KUKA KRL program: ab_com_02_st01_g01.src, ab_com_02_st01_g01.dat

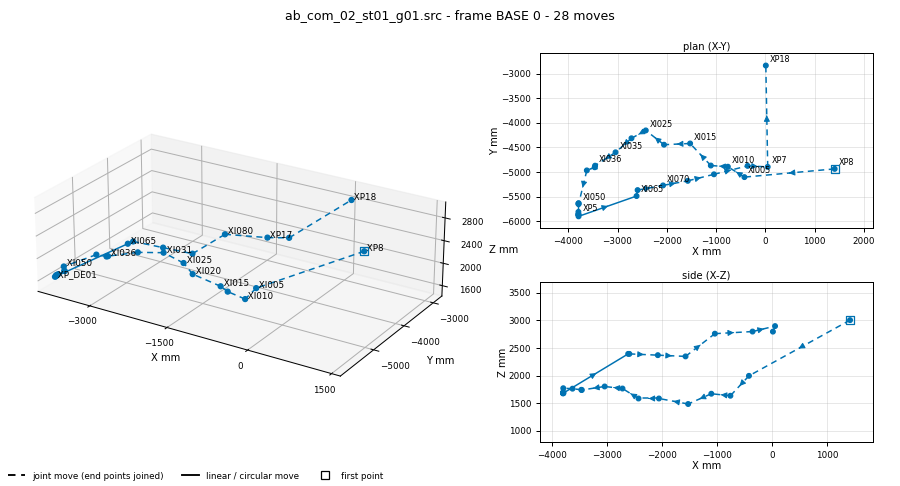
[picture p0: tool path of ab_com_02_st01_g01.src in frame BASE 0, 28 of 28 moves have a stored position in this frame; points joined in program order, loops and branches not executed]
--- ab_com_02_st01_g01.src ---
&ACCESS RVO4
&REL 783
&COMMENT Deposita axor atego 903 geo
&PARAM DISKPATH = KRC:\R1\Program\MANIPULACAO NTC
&PARAM TEMPLATE = C:\KRC\Roboter\Template\vorgabe
&PARAM EDITMASK = *
DEF AB_COM_02_ST01_G01 ( )
;FOLD INI
  ;FOLD BASISTECH INI
    GLOBAL INTERRUPT DECL 3 WHEN $STOPMESS==TRUE DO IR_STOPM ( )
    INTERRUPT ON 3
    BAS (#INITMOV,0)
  ;ENDFOLD (BASISTECH INI)
;FOLD GRIPPERTECH INI
USER_GRP(0,DUMMY,DUMMY,GDEFAULT)
;ENDFOLD (GRIPPERTECH INI)
  ;FOLD USER INI
    ;Make your modifications here

  ;ENDFOLD (USER INI)
;ENDFOLD (INI)

; Caracterizacao dos meios de producao
; Changes: Deposita Traseira LTA/LTB
; Versao Atual: 05/01/2016
; Ferramenta: Gripper 903
; Name: P13.050-R1

chk_w9_wechs_ok ( ) ;CHECK GRIPPER 903

;FOLD PTP P8 Vel=50 % PDAT7 Tool[10]:Grp 903 c/ pc Base[0];%{PE}%R 8.2.20,%MKUKATPBASIS,%CMOVE,%VPTP,%P 1:PTP, 2:P8, 3:, 5:50, 7:PDAT7
$BWDSTART=FALSE
PDAT_ACT=PPDAT7
FDAT_ACT=FP8
BAS(#PTP_PARAMS,50)
PTP XP8
;ENDFOLD

; LIGA INTERTRAVAMENTO 2 C/ R2 GARRA
;FOLD Collision.Monitoring_2_On ;%{PE}%MKUKATPUSER
COLLSTOP( 2, 1 ) ;Interrupt-Controlled
;ENDFOLD

; LIGA INTERTRAVAMENTO 3 C/ R3 GARRA
;FOLD Collision.Monitoring_3_On ;%{PE}%MKUKATPUSER
COLLSTOP( 3, 1 ) ;Interrupt-Controlled
;ENDFOLD

; LIGA INTERTRAVAMENTO 4 C/ R4 GARRA
;FOLD Collision.Monitoring_4_On ;%{PE}%MKUKATPUSER
COLLSTOP( 4, 1 ) ;Interrupt-Controlled
;ENDFOLD

; LIGA INTERTRAVAMENTO 5 C/ R5 GARRA
;FOLD Collision.Monitoring_5_On ;%{PE}%MKUKATPUSER
COLLSTOP( 5, 1 ) ;not Interrupt-Controlled
;ENDFOLD


;FOLD PTP l005 CONT Vel=50 % P_OLP2 Tool[10]:Grp 903 c/ pc Base[0];%{PE}%R 8.2.20,%MKUKATPBASIS,%CMOVE,%VPTP,%P 1:PTP, 2:l005, 3:C_DIS, 5:50, 7:P_OLP2
$BWDSTART=FALSE
PDAT_ACT=PP_OLP2
FDAT_ACT=Fl005
BAS(#PTP_PARAMS,50)
PTP Xl005 C_DIS
;ENDFOLD
;FOLD PTP l010 CONT Vel=50 % P_OLP3 Tool[10]:Grp 903 c/ pc Base[0];%{PE}%R 8.2.20,%MKUKATPBASIS,%CMOVE,%VPTP,%P 1:PTP, 2:l010, 3:C_DIS, 5:50, 7:P_OLP3
$BWDSTART=FALSE
PDAT_ACT=PP_OLP3
FDAT_ACT=Fl010
BAS(#PTP_PARAMS,50)
PTP Xl010 C_DIS
;ENDFOLD

;AGUARDA LIBERACAO DE ENTRADA
;FOLD OUT 3348 'Fora area GEOBOX' State=TRUE ;%{PE}%R 8.2.20,%MKUKATPBASIS,%COUT,%VOUTX,%P 2:3348, 3:Fora area GEOBOX, 5:TRUE, 6:
$OUT[3348]=TRUE
;ENDFOLD
;FOLD OUT 3369 'RB -PLC Interlock' State=TRUE ;%{PE}%R 8.2.20,%MKUKATPBASIS,%COUT,%VOUTX,%P 2:3369, 3:RB -PLC Interlock, 5:TRUE, 6:
$OUT[3369]=TRUE
;ENDFOLD
;FOLD WAIT FOR ( IN 3369 'RB-PLC interlocks' );%{PE}%R 8.2.20,%MKUKATPBASIS,%CEXT_WAIT_FOR,%VEXT_WAIT_FOR,%P 2:, 4:, 5:$IN, 6:3369, 7:RB-PLC interlocks, 9:
WAIT FOR  ( $IN[3369] )
;ENDFOLD
;FOLD OUT 3369 'RB -PLC Interlock' State=FALSE ;%{PE}%R 8.2.20,%MKUKATPBASIS,%COUT,%VOUTX,%P 2:3369, 3:RB -PLC Interlock, 5:FALSE, 6:
$OUT[3369]=FALSE
;ENDFOLD
;FOLD OUT 3348 'Fora area GEOBOX' State=FALSE ;%{PE}%R 8.2.20,%MKUKATPBASIS,%COUT,%VOUTX,%P 2:3348, 3:Fora area GEOBOX, 5:FALSE, 6:
$OUT[3348]=FALSE
;ENDFOLD

;FOLD PTP pp1 CONT Vel=50 % PDAT4 Tool[10]:Grp 903 c/ pc Base[0];%{PE}%R 8.2.20,%MKUKATPBASIS,%CMOVE,%VPTP,%P 1:PTP, 2:pp1, 3:C_DIS, 5:50, 7:PDAT4
$BWDSTART=FALSE
PDAT_ACT=PPDAT4
FDAT_ACT=Fpp1
BAS(#PTP_PARAMS,50)
PTP Xpp1 C_DIS
;ENDFOLD
;FOLD PTP l015 CONT Vel=50 % P_OLP4 Tool[10]:Grp 903 c/ pc Base[0];%{PE}%R 8.2.20,%MKUKATPBASIS,%CMOVE,%VPTP,%P 1:PTP, 2:l015, 3:C_DIS, 5:50, 7:P_OLP4
$BWDSTART=FALSE
PDAT_ACT=PP_OLP4
FDAT_ACT=Fl015
BAS(#PTP_PARAMS,50)
PTP Xl015 C_DIS
;ENDFOLD
;FOLD PTP l020 CONT Vel=50 % P_OLP5 Tool[10]:Grp 903 c/ pc Base[0];%{PE}%R 8.2.20,%MKUKATPBASIS,%CMOVE,%VPTP,%P 1:PTP, 2:l020, 3:C_DIS, 5:50, 7:P_OLP5
$BWDSTART=FALSE
PDAT_ACT=PP_OLP5
FDAT_ACT=Fl020
BAS(#PTP_PARAMS,50)
PTP Xl020 C_DIS
;ENDFOLD
;FOLD PTP l025 CONT Vel=50 % P_OLP6 Tool[10]:Grp 903 c/ pc Base[0];%{PE}%R 8.2.20,%MKUKATPBASIS,%CMOVE,%VPTP,%P 1:PTP, 2:l025, 3:C_DIS, 5:50, 7:P_OLP6
$BWDSTART=FALSE
PDAT_ACT=PP_OLP6
FDAT_ACT=Fl025
BAS(#PTP_PARAMS,50)
PTP Xl025 C_DIS
;ENDFOLD
;FOLD PTP l031 CONT Vel=50 % P_OLP15 Tool[10]:Grp 903 c/ pc Base[0];%{PE}%R 8.2.20,%MKUKATPBASIS,%CMOVE,%VPTP,%P 1:PTP, 2:l031, 3:C_DIS, 5:50, 7:P_OLP15
$BWDSTART=FALSE
PDAT_ACT=PP_OLP15
FDAT_ACT=Fl031
BAS(#PTP_PARAMS,50)
PTP Xl031 C_DIS
;ENDFOLD
;FOLD PTP l035 CONT Vel=50 % P_OLP8 Tool[10]:Grp 903 c/ pc Base[0];%{PE}%R 8.2.20,%MKUKATPBASIS,%CMOVE,%VPTP,%P 1:PTP, 2:l035, 3:C_DIS, 5:50, 7:P_OLP8
$BWDSTART=FALSE
PDAT_ACT=PP_OLP8
FDAT_ACT=Fl035
BAS(#PTP_PARAMS,50)
PTP Xl035 C_DIS
;ENDFOLD
;FOLD PTP l036 CONT Vel=50 % P_OLP16 Tool[10]:Grp 903 c/ pc Base[0];%{PE}%R 8.2.20,%MKUKATPBASIS,%CMOVE,%VPTP,%P 1:PTP, 2:l036, 3:C_DIS, 5:50, 7:P_OLP16
$BWDSTART=FALSE
PDAT_ACT=PP_OLP16
FDAT_ACT=Fl036
BAS(#PTP_PARAMS,50)
PTP Xl036 C_DIS
;ENDFOLD

;AGUARDA LIBERACAO PARA DEPOSITO
;FOLD OUT 3374 'Lib. Dep. Axor/Atego' State=TRUE ;%{PE}%R 8.2.20,%MKUKATPBASIS,%COUT,%VOUTX,%P 2:3374, 3:Lib. Dep. Axor/Atego, 5:TRUE, 6:
$OUT[3374]=TRUE
;ENDFOLD
;FOLD OUT 3372 'Lib. pré Dep. Axor/Atego' State=TRUE ;%{PE}%R 8.2.20,%MKUKATPBASIS,%COUT,%VOUTX,%P 2:3372, 3:Lib. pré Dep. Axor/Atego, 5:TRUE, 6:
$OUT[3372]=TRUE
;ENDFOLD
;FOLD WAIT FOR ( IN 3372 'Lib. pré Deposito Axor/Atego' );%{PE}%R 8.2.20,%MKUKATPBASIS,%CEXT_WAIT_FOR,%VEXT_WAIT_FOR,%P 2:, 4:, 5:$IN, 6:3372, 7:Lib. pré Deposito Axor/Atego, 9:
WAIT FOR  ( $IN[3372] )
;ENDFOLD
;FOLD OUT 3372 'Lib. pré Dep. Axor/Atego' State=FALSE ;%{PE}%R 8.2.20,%MKUKATPBASIS,%COUT,%VOUTX,%P 2:3372, 3:Lib. pré Dep. Axor/Atego, 5:FALSE, 6:
$OUT[3372]=FALSE
;ENDFOLD
;FOLD OUT 3374 'Lib. Dep. Axor/Atego' State=FALSE ;%{PE}%R 8.2.20,%MKUKATPBASIS,%COUT,%VOUTX,%P 2:3374, 3:Lib. Dep. Axor/Atego, 5:FALSE, 6:
$OUT[3374]=FALSE
;ENDFOLD

;FOLD PTP l040 CONT Vel=50 % P_OLP9 Tool[10]:Grp 903 c/ pc Base[0];%{PE}%R 8.2.20,%MKUKATPBASIS,%CMOVE,%VPTP,%P 1:PTP, 2:l040, 3:C_DIS, 5:50, 7:P_OLP9
$BWDSTART=FALSE
PDAT_ACT=PP_OLP9
FDAT_ACT=Fl040
BAS(#PTP_PARAMS,50)
PTP Xl040 C_DIS
;ENDFOLD
;FOLD PTP l045 CONT Vel=50 % PDAT1 Tool[10]:Grp 903 c/ pc Base[0];%{PE}%R 8.2.20,%MKUKATPBASIS,%CMOVE,%VPTP,%P 1:PTP, 2:l045, 3:C_DIS, 5:50, 7:PDAT1
$BWDSTART=FALSE
PDAT_ACT=PPDAT1
FDAT_ACT=Fl045
BAS(#PTP_PARAMS,50)
PTP Xl045 C_DIS
;ENDFOLD

; POSICAO DE VERIFICACAO DE VENTOSA OK
;FOLD PTP l050 Vel=50 % P_OLP10 Tool[10]:Grp 903 c/ pc Base[0];%{PE}%R 8.2.20,%MKUKATPBASIS,%CMOVE,%VPTP,%P 1:PTP, 2:l050, 3:, 5:50, 7:P_OLP10
$BWDSTART=FALSE
PDAT_ACT=PP_OLP10
FDAT_ACT=Fl050
BAS(#PTP_PARAMS,50)
PTP Xl050
;ENDFOLD

IF (NOT(GHOST())) THEN
chk_w9_grp5_vac_on( )      ; VENTOSA OK
ENDIF

;FOLD PTP pp2 CONT Vel=100 % PDAT5 Tool[10]:Grp 903 c/ pc Base[0];%{PE}%R 8.2.20,%MKUKATPBASIS,%CMOVE,%VPTP,%P 1:PTP, 2:pp2, 3:C_DIS, 5:100, 7:PDAT5
$BWDSTART=FALSE
PDAT_ACT=PPDAT5
FDAT_ACT=Fpp2
BAS(#PTP_PARAMS,100)
PTP Xpp2 C_DIS
;ENDFOLD
;FOLD PTP l055 CONT Vel=100 % P_OLP11 Tool[10]:Grp 903 c/ pc Base[0];%{PE}%R 8.2.20,%MKUKATPBASIS,%CMOVE,%VPTP,%P 1:PTP, 2:l055, 3:C_DIS, 5:100, 7:P_OLP11
$BWDSTART=FALSE
PDAT_ACT=PP_OLP11
FDAT_ACT=Fl055
BAS(#PTP_PARAMS,100)
PTP Xl055 C_DIS
;ENDFOLD
;FOLD LIN P9 CONT Vel=0.5 m/s CPDAT8 Tool[10]:Grp 903 c/ pc Base[0];%{PE}%R 8.2.20,%MKUKATPBASIS,%CMOVE,%VLIN,%P 1:LIN, 2:P9, 3:C_DIS C_DIS, 5:0.5, 7:CPDAT8
$BWDSTART=FALSE
LDAT_ACT=LCPDAT8
FDAT_ACT=FP9
BAS(#CP_PARAMS,0.5)
LIN XP9 C_DIS C_DIS
;ENDFOLD

; ABRE GRAMPOS INFERIORES P/ ENCAIXAR NA GEOBOX
; TECLA DE ESTADO "7"
;FOLD SET Z1.1/2 GRP AXOR 903 State=OPN GDAT1;%{PE}%R 8.2.1,%MKUKATPGRP,%CGRP,%VGRP,%P 2:7, 4:1, 5:#NO, 6:GDAT1, 8:0, 10:0
H50(GRP,7,1,GGDAT1)
;ENDFOLD
chk_w9_grp1_opn( )

;FOLD LIN P5 CONT Vel=0.5 m/s CPDAT4 Tool[10]:Grp 903 c/ pc Base[0];%{PE}%R 8.2.20,%MKUKATPBASIS,%CMOVE,%VLIN,%P 1:LIN, 2:P5, 3:C_DIS C_DIS, 5:0.5, 7:CPDAT4
$BWDSTART=FALSE
LDAT_ACT=LCPDAT4
FDAT_ACT=FP5
BAS(#CP_PARAMS,0.5)
LIN XP5 C_DIS C_DIS
;ENDFOLD
;FOLD LIN P14 CONT Vel=0.5 m/s CPDAT13 Tool[10]:Grp 903 c/ pc Base[0];%{PE}%R 8.2.20,%MKUKATPBASIS,%CMOVE,%VLIN,%P 1:LIN, 2:P14, 3:C_DIS C_DIS, 5:0.5, 7:CPDAT13
$BWDSTART=FALSE
LDAT_ACT=LCPDAT13
FDAT_ACT=FP14
BAS(#CP_PARAMS,0.5)
LIN XP14 C_DIS C_DIS
;ENDFOLD

; POSICAO DE APOIO ROLETE
;FOLD LIN P12 Vel=0.3 m/s CPDAT11 Tool[10]:Grp 903 c/ pc Base[0];%{PE}%R 8.2.20,%MKUKATPBASIS,%CMOVE,%VLIN,%P 1:LIN, 2:P12, 3:, 5:0.3, 7:CPDAT11
$BWDSTART=FALSE
LDAT_ACT=LCPDAT11
FDAT_ACT=FP12
BAS(#CP_PARAMS,0.3)
LIN XP12
;ENDFOLD

; DESLIGA INTERTRAVAMENTO 3 C/ R3 GARRA
;FOLD Collision.Monitoring_3_Off . ;%{PE}%MKUKATPUSER
COLLSTOP( 3, 2+0 )
;ENDFOLD

; DESLIGA INTERTRAVAMENTO 5 C/ R5 GARRA
;FOLD Collision.Monitoring_5_Off . ;%{PE}%MKUKATPUSER
COLLSTOP( 5, 2+0 )
;ENDFOLD

;FOLD ; Aguarda posicionamento dos Grippers R2 e R3 com rolamentos;%{PE}%R 8.2.20,%MKUKATPBASIS,%CCOMMENT,%VNORMAL,%P 2:Aguarda posicionamento dos Grippers R2 e R3 com rolamentos
;ENDFOLD
;FOLD OUT 3373 'Em pos de pre Dep AXOR/ATEGO' State=TRUE ;%{PE}%R 8.2.20,%MKUKATPBASIS,%COUT,%VOUTX,%P 2:3373, 3:Em pos de pre Dep AXOR/ATEGO, 5:TRUE, 6:
$OUT[3373]=TRUE
;ENDFOLD
;FOLD WAIT FOR ( IN 3374 'Lib. Deposito Axor/Atego' );%{PE}%R 8.2.20,%MKUKATPBASIS,%CEXT_WAIT_FOR,%VEXT_WAIT_FOR,%P 2:, 4:, 5:$IN, 6:3374, 7:Lib. Deposito Axor/Atego, 9:
WAIT FOR  ( $IN[3374] )
;ENDFOLD
;FOLD OUT 3373 'Em pos de pre Dep AXOR/ATEGO' State=FALSE ;%{PE}%R 8.2.20,%MKUKATPBASIS,%COUT,%VOUTX,%P 2:3373, 3:Em pos de pre Dep AXOR/ATEGO, 5:FALSE, 6:
$OUT[3373]=FALSE
;ENDFOLD

;FOLD ; Desliga Ventosa / Recua Cilindros / Verifica;%{PE}%R 8.2.20,%MKUKATPBASIS,%CCOMMENT,%VNORMAL,%P 2:Desliga Ventosa / Recua Cilindros / Verifica
;ENDFOLD
;FOLD SET Z6.1 VAC AXOR 903 State=BLOW GDAT26;%{PE}%R 8.2.1,%MKUKATPGRP,%CGRP,%VGRP,%P 2:13, 4:2, 5:#NO, 6:GDAT26, 8:0, 10:0
H50(GRP,13,2,GGDAT26)
;ENDFOLD
;FOLD SET Z6.1 VAC AXOR 903 State=OFF GDAT6;%{PE}%R 8.2.1,%MKUKATPGRP,%CGRP,%VGRP,%P 2:13, 4:3, 5:#NO, 6:GDAT6, 8:0, 10:0
H50(GRP,13,3,GGDAT6)
;ENDFOLD
;FOLD SET Z7.1 GRP 7 AXOR 903 State=OPN GDAT28;%{PE}%R 8.2.1,%MKUKATPGRP,%CGRP,%VGRP,%P 2:14, 4:1, 5:#NO, 6:GDAT28, 8:0, 10:0
H50(GRP,14,1,GGDAT28)
;ENDFOLD
chk_w9_grp4_opn( )
chk_w9_grp5_vac_off( )

; POSICAO DE DEPOSITO LTA/LTB
;FOLD LIN P_DE01  Vel=0.25 m/s L_OLP3 Tool[10]:Grp 903 c/ pc Base[0];%{PE}%R8.2.19,%MKUKATPBASIS,%CMOVE,%VLIN,%P 1:LIN, 2:P_DE01, 3: , 5:0.25, 7:L_OLP3
$BWDSTART = FALSE
LDAT_ACT= LL_OLP3
FDAT_ACT= FP_DE01
BAS(#CP_PARAMS,0.25)
LIN XP_DE01
;ENDFOLD

; DESLIGA INTERTRAVAMENTO 4 C/ R4 GARRA
;FOLD Collision.Monitoring_4_Off . ;%{PE}%MKUKATPUSER
COLLSTOP( 4, 2+0 )
;ENDFOLD

;FOLD OUT 3375 'Lib. p/ sair s/ Gripper Axor/Atego' State=TRUE ;%{PE}%R 8.2.20,%MKUKATPBASIS,%COUT,%VOUTX,%P 2:3375, 3:Lib. p/ sair s/ Gripper Axor/Atego, 5:TRUE, 6:
$OUT[3375]=TRUE
;ENDFOLD

; FECHA GRAMPOS INFERIORES
; TECLA DE ESTADO "7"
;FOLD SET Z1.1/2 GRP AXOR 903 State=CLO GDAT5;%{PE}%R 8.2.1,%MKUKATPGRP,%CGRP,%VGRP,%P 2:7, 4:2, 5:#NO, 6:GDAT5, 8:0, 10:0
H50(GRP,7,2,GGDAT5)
;ENDFOLD
chk_w9_grp1_clo( )

;AGUARDA LIBERACAO SAIR SEM GARRA
;FOLD OUT 3375 'Lib. p/ sair s/ Gripper Axor/Atego' State=TRUE ;%{PE}%R 8.2.20,%MKUKATPBASIS,%COUT,%VOUTX,%P 2:3375, 3:Lib. p/ sair s/ Gripper Axor/Atego, 5:TRUE, 6:
$OUT[3375]=TRUE
;ENDFOLD
;FOLD WAIT FOR ( IN 3375 'Lib. p/ sair s/ Gripper Axor/Atego' );%{PE}%R 8.2.20,%MKUKATPBASIS,%CEXT_WAIT_FOR,%VEXT_WAIT_FOR,%P 2:, 4:, 5:$IN, 6:3375, 7:Lib. p/ sair s/ Gripper Axor/Atego, 9:
WAIT FOR  ( $IN[3375] )
;ENDFOLD
;FOLD OUT 3375 'Lib. p/ sair s/ Gripper Axor/Atego' State=FALSE ;%{PE}%R 8.2.20,%MKUKATPBASIS,%COUT,%VOUTX,%P 2:3375, 3:Lib. p/ sair s/ Gripper Axor/Atego, 5:FALSE, 6:
$OUT[3375]=FALSE
;ENDFOLD

; COMANDOS PARA DESACOPLAR GRIPPER
;FOLD OUT 224 'Bloquear MPS' State=FALSE ;%{PE}%R 8.2.20,%MKUKATPBASIS,%COUT,%VOUTX,%P 2:224, 3:Bloquear MPS, 5:FALSE, 6:
$OUT[224]=FALSE
;ENDFOLD
;FOLD OUT 223 'Desbloquear MPS' State=TRUE ;%{PE}%R 8.2.20,%MKUKATPBASIS,%COUT,%VOUTX,%P 2:223, 3:Desbloquear MPS, 5:TRUE, 6:
$OUT[223]=TRUE
;ENDFOLD
;FOLD WAIT FOR ( IN 217 'MPS Destravado' );%{PE}%R 8.2.20,%MKUKATPBASIS,%CEXT_WAIT_FOR,%VEXT_WAIT_FOR,%P 2:, 4:, 5:$IN, 6:217, 7:MPS Destravado, 9:
WAIT FOR  ( $IN[217] )
;ENDFOLD
;FOLD WAIT FOR NOT ( IN 221 'MPS Travado' );%{PE}%R 8.2.20,%MKUKATPBASIS,%CEXT_WAIT_FOR,%VEXT_WAIT_FOR,%P 2:NOT, 4:, 5:$IN, 6:221, 7:MPS Travado, 9:
WAIT FOR  NOT ( $IN[221] )
;ENDFOLD
;FOLD WAIT Time=0.5 sec;%{PE}%R 8.2.20,%MKUKATPBASIS,%CWAIT,%VWAIT,%P 3:0.5
WAIT SEC 0.5
;ENDFOLD
;FOLD IBUS OFF;%{PE}%R 8.2.20,%MKUKATPBASIS,%CIBUS,%VMAP,%P 2:#OFF, 3:1
$IBUS_OFF=$IBUS_ON
$IBUS_ON=0
;ENDFOLD
;FOLD WAIT Time=0.25 sec;%{PE}%R 8.2.20,%MKUKATPBASIS,%CWAIT,%VWAIT,%P 3:0.25
WAIT SEC 0.25
;ENDFOLD

;FOLD LIN l065 Vel=0.25 m/s L_OLP4 Tool[8]:TOOL_CHANGER Base[0];%{PE}%R 8.2.20,%MKUKATPBASIS,%CMOVE,%VLIN,%P 1:LIN, 2:l065, 3:, 5:0.25, 7:L_OLP4
$BWDSTART=FALSE
LDAT_ACT=LL_OLP4
FDAT_ACT=Fl065
BAS(#CP_PARAMS,0.25)
LIN Xl065
;ENDFOLD

;FOLD WAIT FOR NOT ( IN 219 'Posicao p/ Acoplamento OK' );%{PE}%R 8.2.20,%MKUKATPBASIS,%CEXT_WAIT_FOR,%VEXT_WAIT_FOR,%P 2:NOT, 4:, 5:$IN, 6:219, 7:Posicao p/ Acoplamento OK, 9:
WAIT FOR  NOT ( $IN[219] )
;ENDFOLD
;FOLD OUT 223 'Desbloquear MPS' State=FALSE ;%{PE}%R 8.2.20,%MKUKATPBASIS,%COUT,%VOUTX,%P 2:223, 3:Desbloquear MPS, 5:FALSE, 6:
$OUT[223]=FALSE
;ENDFOLD

;FOLD LIN P2 CONT Vel=1 m/s CPDAT1 Tool[10]:Grp 903 c/ pc Base[0];%{PE}%R 8.2.20,%MKUKATPBASIS,%CMOVE,%VLIN,%P 1:LIN, 2:P2, 3:C_DIS C_DIS, 5:1, 7:CPDAT1
$BWDSTART=FALSE
LDAT_ACT=LCPDAT1
FDAT_ACT=FP2
BAS(#CP_PARAMS,1)
LIN XP2 C_DIS C_DIS
;ENDFOLD
;FOLD PTP l070 CONT Vel=100 % P_OLP12 Tool[10]:Grp 903 c/ pc Base[0];%{PE}%R 8.2.20,%MKUKATPBASIS,%CMOVE,%VPTP,%P 1:PTP, 2:l070, 3:C_DIS, 5:100, 7:P_OLP12
$BWDSTART=FALSE
PDAT_ACT=PP_OLP12
FDAT_ACT=Fl070
BAS(#PTP_PARAMS,100)
PTP Xl070 C_DIS
;ENDFOLD
;FOLD PTP l075 CONT Vel=100 % P_OLP13 Tool[10]:Grp 903 c/ pc Base[0];%{PE}%R 8.2.20,%MKUKATPBASIS,%CMOVE,%VPTP,%P 1:PTP, 2:l075, 3:C_DIS, 5:100, 7:P_OLP13
$BWDSTART=FALSE
PDAT_ACT=PP_OLP13
FDAT_ACT=Fl075
BAS(#PTP_PARAMS,100)
PTP Xl075 C_DIS
;ENDFOLD
;FOLD PTP l080 CONT Vel=100 % P_OLP14 Tool[10]:Grp 903 c/ pc Base[0];%{PE}%R 8.2.20,%MKUKATPBASIS,%CMOVE,%VPTP,%P 1:PTP, 2:l080, 3:C_DIS, 5:100, 7:P_OLP14
$BWDSTART=FALSE
PDAT_ACT=PP_OLP14
FDAT_ACT=Fl080
BAS(#PTP_PARAMS,100)
PTP Xl080 C_DIS
;ENDFOLD
;FOLD PTP P17 CONT Vel=100 % PDAT10 Tool[10]:Grp 903 c/ pc Base[0];%{PE}%R 8.2.20,%MKUKATPBASIS,%CMOVE,%VPTP,%P 1:PTP, 2:P17, 3:C_DIS, 5:100, 7:PDAT10
$BWDSTART=FALSE
PDAT_ACT=PPDAT10
FDAT_ACT=FP17
BAS(#PTP_PARAMS,100)
PTP XP17 C_DIS
;ENDFOLD

; DESLIGA INTERTRAVAMENTO 2 C/ R2 GARRA
;FOLD Collision.Monitoring_2_Off . ;%{PE}%MKUKATPUSER
COLLSTOP( 2, 2+0 )
;ENDFOLD

;LIBERA AREA
;FOLD OUT 3348 'Fora area GEOBOX' State=TRUE ;%{PE}%R 8.2.20,%MKUKATPBASIS,%COUT,%VOUTX,%P 2:3348, 3:Fora area GEOBOX, 5:TRUE, 6:
$OUT[3348]=TRUE
;ENDFOLD
;FOLD PULSE 3344 'R1 Entregou Peça GeoBox' State=TRUE Time=3 sec;%{PE}%R 8.2.20,%MKUKATPBASIS,%COUT,%VPULSE,%P 2:3344, 3:R1 Entregou Peça GeoBox, 5:TRUE, 6:, 8:3
PULSE($OUT[3344], TRUE,3)
;ENDFOLD

;FOLD PTP P7 CONT Vel=100 % PDAT6 Tool[10]:Grp 903 c/ pc Base[0];%{PE}%R 8.2.20,%MKUKATPBASIS,%CMOVE,%VPTP,%P 1:PTP, 2:P7, 3:C_DIS, 5:100, 7:PDAT6
$BWDSTART=FALSE
PDAT_ACT=PPDAT6
FDAT_ACT=FP7
BAS(#PTP_PARAMS,100)
PTP XP7 C_DIS
;ENDFOLD
;FOLD PTP P18 CONT Vel=100 % PDAT11 Tool[10]:Grp 903 c/ pc Base[0];%{PE}%R 8.2.20,%MKUKATPBASIS,%CMOVE,%VPTP,%P 1:PTP, 2:P18, 3:C_DIS, 5:100, 7:PDAT11
$BWDSTART=FALSE
PDAT_ACT=PPDAT11
FDAT_ACT=FP18
BAS(#PTP_PARAMS,100)
PTP XP18 C_DIS
;ENDFOLD

END

--- ab_com_02_st01_g01.dat ---
&ACCESS RVO4
&REL 783
&COMMENT Deposita axor atego 903 geo
&PARAM DISKPATH = KRC:\R1\Program\MANIPULACAO NTC
&PARAM TEMPLATE = C:\KRC\Roboter\Template\vorgabe
&PARAM EDITMASK = *
DEFDAT  ab_com_02_st01_g01
;FOLD EXTERNAL DECLARATIONS;%{PE}%MKUKATPBASIS,%CEXT,%VCOMMON,%P
;FOLD GRIPPERTECH EXT
EXT  H50 (INT  :IN,INT  :IN,INT  :IN,GRP_TYP  :IN )
;ENDFOLD (GRIPPERTECH EXT)
;FOLD SPOTTECH EXT

;ENDFOLD (SPOTTECH EXT)
;FOLD BASISTECH EXT;%{PE}%MKUKATPBASIS,%CEXT,%VEXT,%P
EXT  BAS (BAS_COMMAND  :IN,REAL  :IN )
DECL INT SUCCESS
;ENDFOLD (BASISTECH EXT)
;FOLD USER EXT;%{E}%MKUKATPUSER,%CEXT,%VEXT,%P
;Make your modifications here

;ENDFOLD (USER EXT)
DECL FDAT Fl005={TOOL_NO 10,BASE_NO 0,IPO_FRAME #BASE,POINT2[] " ",TQ_STATE FALSE}
DECL PDAT PP_OLP2={VEL 100.0,ACC 50.0,APO_DIST 30.0,APO_MODE #CDIS}
DECL E6POS Xl005={X -423.688995,Y -5102.93994,Z 1996.18701,A -23.8787003,B 72.4475021,C 42.6447983,S 6,T 50,E1 -2500.0,E2 0.0,E3 0.0,E4 0.0,E5 0.0,E6 0.0}
DECL FDAT Fl010={TOOL_NO 10,BASE_NO 0,IPO_FRAME #BASE,POINT2[] " "}
DECL PDAT PP_OLP3={VEL 100.0,ACC 50.0,APO_DIST 30.0,APO_MODE #CDIS}
DECL E6POS Xl010={X -760.000977,Y -4891.79297,Z 1635.40405,A 7.58529997,B 87.1332016,C 85.2861023,S 6,T 26,E1 -2800.0,E2 0.0,E3 0.0,E4 0.0,E5 0.0,E6 0.0}
DECL FDAT Fl015={TOOL_NO 10,BASE_NO 0,IPO_FRAME #BASE,POINT2[] " "}
DECL PDAT PP_OLP4={VEL 100.0,ACC 50.0,APO_DIST 30.0,APO_MODE #CDIS}
DECL E6POS Xl015={X -1525.96594,Y -4420.06396,Z 1485.40295,A -15.7344999,B 87.1332016,C 85.2856979,S 6,T 26,E1 -2800.0,E2 0.0,E3 0.0,E4 0.0,E5 0.0,E6 0.0}
DECL FDAT Fl020={TOOL_NO 10,BASE_NO 0,IPO_FRAME #BASE,POINT2[] " "}
DECL PDAT PP_OLP5={VEL 100.0,ACC 50.0,APO_DIST 30.0,APO_MODE #CDIS}
DECL E6POS Xl020={X -2055.78906,Y -4445.21289,Z 1585.40198,A -17.4160004,B 87.1333008,C 85.2846985,S 6,T 50,E1 -3000.0,E2 0.0,E3 0.0,E4 0.0,E5 0.0,E6 0.0}
DECL FDAT Fl025={TOOL_NO 10,BASE_NO 0,IPO_FRAME #BASE,POINT2[] " "}
DECL PDAT PP_OLP6={VEL 100.0,ACC 50.0,APO_DIST 30.0,APO_MODE #CDIS}
DECL E6POS Xl025={X -2426.0979,Y -4154.93311,Z 1585.40198,A -37.4154015,B 87.1333008,C 85.2853012,S 6,T 50,E1 -3500.0,E2 0.0,E3 0.0,E4 0.0,E5 0.0,E6 0.0}
DECL FDAT Fl030={TOOL_NO 10,BASE_NO 0,IPO_FRAME #BASE,POINT2[] " "}
DECL PDAT PP_OLP7={VEL 100.0,ACC 50.0,APO_DIST 30.0,APO_MODE #CDIS}
DECL E6POS Xl030={X -2639.52393,Y -4314.86084,Z 1766.01404,A -99.9337006,B 83.2399979,C 22.9171009,S 6,T 50,E1 -3600.0,E2 0.0,E3 0.0,E4 0.0,E5 0.0,E6 0.0}
DECL FDAT Fl035={TOOL_NO 10,BASE_NO 0,IPO_FRAME #BASE,POINT2[] " "}
DECL PDAT PP_OLP8={VEL 100.0,ACC 50.0,APO_DIST 30.0,APO_MODE #CDIS}
DECL E6POS Xl035={X -3040.146,Y -4599.22119,Z 1803.30896,A -99.9337997,B 83.2399979,C 22.9169998,S 6,T 50,E1 -4500.0,E2 0.0,E3 0.0,E4 0.0,E5 0.0,E6 0.0}
DECL FDAT Fl040={TOOL_NO 10,BASE_NO 0,IPO_FRAME #BASE,POINT2[] " "}
DECL PDAT PP_OLP9={VEL 100.0,ACC 50.0,APO_DIST 20.0,APO_MODE #CDIS}
DECL E6POS Xl040={X -3462.30005,Y -4903.24805,Z 1743.26099,A -94.3171768,B 83.0381165,C 8.50555897,S 6,T 50,E1 -4500.0,E2 0.0,E3 0.0,E4 0.0,E5 0.0,E6 0.0}
DECL FDAT Fl045={TOOL_NO 10,BASE_NO 0,IPO_FRAME #BASE,POINT2[] " ",TQ_STATE FALSE}
DECL E6POS Xl045={X -3622.87012,Y -4966.85986,Z 1763.39001,A -93.2050934,B 83.0319366,C 5.76104593,S 6,T 50,E1 -4448.65479,E2 0.0,E3 0.0,E4 0.0,E5 0.0,E6 0.0}
DECL FDAT Fl050={TOOL_NO 10,BASE_NO 0,IPO_FRAME #BASE,POINT2[] " "}
DECL PDAT PP_OLP10={VEL 100.0,ACC 50.0,APO_DIST 20.0,APO_MODE #CDIS}
DECL E6POS Xl050={X -3790.37305,Y -5652.16406,Z 1771.51599,A -89.9828186,B 79.9307404,C -1.746503,S 6,T 50,E1 -4600.0,E2 0.0,E3 0.0,E4 0.0,E5 0.0,E6 0.0}
DECL FDAT Fl055={TOOL_NO 10,BASE_NO 0,IPO_FRAME #BASE,POINT2[] " "}
DECL PDAT PP_OLP11={VEL 100.0,ACC 50.0,APO_DIST 10.0,APO_MODE #CDIS}
DECL E6POS Xl055={X -3788.71802,Y -5632.47705,Z 1681.61902,A -168.600601,B 89.5499115,C -80.7964172,S 6,T 50,E1 -4900.00098,E2 0.0,E3 0.0,E4 0.0,E5 0.0,E6 0.0}
DECL FDAT FP_DE01={TOOL_NO 10,BASE_NO 0,IPO_FRAME #BASE,POINT2[] " "}
DECL E6POS XP_DE01={X -3790.427,Y -5899.54883,Z 1682.755,A -161.369598,B 89.5251999,C -73.5557632,S 6,T 50,E1 -4900.00195,E2 0.0,E3 0.0,E4 0.0,E5 0.0,E6 0.0}
DECL LDAT LL_OLP3={VEL 0.25,ACC 100.0,APO_DIST 0.0,APO_FAC 0.0,ORI_TYP #VAR,CIRC_TYP #BASE,JERK_FAC 50.0}
DECL FDAT Fl065={TOOL_NO 8,BASE_NO 0,IPO_FRAME #BASE,POINT2[] " ",TQ_STATE FALSE}
DECL E6POS Xl065={X -2613.11694,Y -5487.26514,Z 2394.53589,A 170.962402,B 75.0736465,C -89.0954132,S 6,T 50,E1 -4900.0542,E2 0.0,E3 0.0,E4 0.0,E5 0.0,E6 0.0}
DECL LDAT LL_OLP4={VEL 0.25,ACC 100.0,APO_DIST 0.0,APO_FAC 0.0,ORI_TYP #VAR,CIRC_TYP #BASE,JERK_FAC 50.0}
DECL FDAT Fl070={TOOL_NO 8,BASE_NO 0,IPO_FRAME #BASE,POINT2[] " ",TQ_STATE FALSE}
DECL PDAT PP_OLP12={VEL 100.0,ACC 100.0,APO_DIST 100.0,APO_MODE #CDIS}
DECL E6POS Xl070={X -2075.48193,Y -5271.26807,Z 2371.01001,A 167.393204,B 75.5991974,C -93.8111496,S 6,T 50,E1 -4835.91016,E2 0.0,E3 0.0,E4 0.0,E5 0.0,E6 0.0}
DECL FDAT Fl075={TOOL_NO 8,BASE_NO 0,IPO_FRAME #BASE,POINT2[] " ",TQ_STATE FALSE}
DECL PDAT PP_OLP13={VEL 100.0,ACC 100.0,APO_DIST 100.0,APO_MODE #CDIS}
DECL E6POS Xl075={X -1573.45398,Y -5178.67822,Z 2348.62988,A 163.685196,B 76.0549622,C -98.6335831,S 6,T 50,E1 -4773.56689,E2 0.0,E3 0.0,E4 0.0,E5 0.0,E6 0.0}
DECL FDAT Fl080={TOOL_NO 8,BASE_NO 0,IPO_FRAME #BASE,POINT2[] " ",TQ_STATE FALSE}
DECL PDAT PP_OLP14={VEL 100.0,ACC 100.0,APO_DIST 100.0,APO_MODE #CDIS}
DECL E6POS Xl080={X -1041.828,Y -5045.97021,Z 2760.61694,A 170.962799,B 21.0511398,C -87.2434464,S 6,T 50,E1 -4398.23193,E2 0.0,E3 0.0,E4 0.0,E5 0.0,E6 0.0}
DECL BASIS_SUGG_T LAST_BASIS={POINT1[] "P21                     ",POINT2[] "P21                     ",CP_PARAMS[] "CPDAT13                 ",PTP_PARAMS[] "PDAT14                  ",CONT[] "C_DIS                   ",CP_VEL[] "0.3                     ",PTP_VEL[] "100                     ",SYNC_PARAMS[] "SYNCDAT                 ",SPL_NAME[] "S0                      "}
DECL PDAT PPDAT1={VEL 100.0,ACC 50.0,APO_DIST 20.0,APO_MODE #CDIS}
DECL GRP_SUGG_T LAST_GRP={NUMBER[] "13                      ",STATE[] "2                       ",PARAMS[] "GDAT6                   "}
DECL GRP_TYP GGDAT1={G_APO #NO,GRP_TIME 0.200000003,CTRL #OFF,DLY 0,DST 1}
DECL GRP_TYP GGDAT2={G_APO #NO,GRP_TIME 0.200000003,CTRL #OFF,DLY 0,DST 1}
DECL E6POS XP2={X -2592.01904,Y -5366.5332,Z 2394.03711,A 170.962494,B 75.0737228,C -89.0953064,S 6,T 50,E1 -4900.0542,E2 0.0,E3 0.0,E4 0.0,E5 0.0,E6 0.0}
DECL FDAT FP2={TOOL_NO 8,BASE_NO 0,IPO_FRAME #BASE,POINT2[] " ",TQ_STATE FALSE}
DECL LDAT LCPDAT1={VEL 2.0,ACC 100.0,APO_DIST 50.0,APO_FAC 50.0,AXIS_VEL 100.0,AXIS_ACC 100.0,ORI_TYP #VAR,CIRC_TYP #BASE,JERK_FAC 50.0,GEAR_JERK 50.0,EXAX_IGN 0}
DECL LDAT LCPDAT4={VEL 2.0,ACC 100.0,APO_DIST 0.0,APO_FAC 50.0,AXIS_VEL 100.0,AXIS_ACC 100.0,ORI_TYP #VAR,CIRC_TYP #BASE,JERK_FAC 50.0,GEAR_JERK 50.0,EXAX_IGN 0}
DECL E6POS XP5={X -3791.41504,Y -5863.64404,Z 1696.83301,A -104.325798,B 88.5755615,C -16.5170307,S 6,T 50,E1 -4900.00293,E2 0.0,E3 0.0,E4 0.0,E5 0.0,E6 0.0}
DECL FDAT FP5={TOOL_NO 10,BASE_NO 0,IPO_FRAME #BASE,POINT2[] " ",TQ_STATE FALSE}
DECL E6POS XPP1={X -1106.04895,Y -4867.78809,Z 1671.68103,A 0.654276073,B 81.7736588,C 85.5849915,S 6,T 26,E1 -2679.30298,E2 0.0,E3 0.0,E4 0.0,E5 0.0,E6 0.0}
DECL FDAT Fpp1={TOOL_NO 10,BASE_NO 0,IPO_FRAME #BASE,POINT2[] " ",TQ_STATE FALSE}
DECL PDAT PPDAT4={VEL 100.0,ACC 50.0,APO_DIST 30.0,APO_MODE #CDIS}
DECL E6POS XPP2={X -3793.92505,Y -5639.02295,Z 1687.98804,A -103.525002,B 88.1913071,C -14.9143295,S 6,T 50,E1 -4850.00781,E2 0.0,E3 0.0,E4 0.0,E5 0.0,E6 0.0}
DECL FDAT Fpp2={TOOL_NO 10,BASE_NO 0,IPO_FRAME #BASE,POINT2[] " ",TQ_STATE FALSE}
DECL PDAT PPDAT5={VEL 100.0,ACC 50.0,APO_DIST 10.0,APO_MODE #CDIS}
DECL E6POS XP7={X 49.3248291,Y -4895.24902,Z 2898.11304,A -21.01828,B -59.8416786,C 116.318901,S 2,T 10,E1 -3482.93408,E2 0.0,E3 0.0,E4 0.0,E5 0.0,E6 0.0}
DECL FDAT FP7={TOOL_NO 8,BASE_NO 0,IPO_FRAME #BASE,POINT2[] " ",TQ_STATE FALSE}
DECL PDAT PPDAT6={VEL 100.0,ACC 100.0,APO_DIST 100.0,APO_MODE #CDIS}
DECL PDAT PPDAT7={VEL 100.0,ACC 100.0,APO_DIST 100.0,APO_MODE #CDIS}
DECL E6POS XP8={X 1408.87598,Y -4935.90723,Z 3006.11108,A -20.0040207,B 69.0891495,C -21.5691395,S 2,T 11,E1 -3220.81396,E2 0.0,E3 0.0,E4 0.0,E5 0.0,E6 0.0}
DECL FDAT FP8={TOOL_NO 10,BASE_NO 0,IPO_FRAME #BASE,POINT2[] " ",TQ_STATE FALSE}
DECL E6POS XP9={X -3793.64307,Y -5809.64111,Z 1692.59399,A -127.257797,B 89.1818085,C -39.4533691,S 6,T 50,E1 -4900.00391,E2 0.0,E3 0.0,E4 0.0,E5 0.0,E6 0.0}
DECL FDAT FP9={TOOL_NO 10,BASE_NO 0,IPO_FRAME #BASE,POINT2[] " ",TQ_STATE FALSE}
DECL LDAT LCPDAT8={VEL 2.0,ACC 100.0,APO_DIST 5.0,APO_FAC 50.0,AXIS_VEL 100.0,AXIS_ACC 100.0,ORI_TYP #VAR,CIRC_TYP #BASE,JERK_FAC 50.0,GEAR_JERK 50.0,EXAX_IGN 0}
DECL E6POS XP12={X -3795.78711,Y -5864.21484,Z 1677.55798,A -147.738907,B 89.548027,C -59.3011093,S 6,T 50,E1 -4886.14795,E2 0.0,E3 0.0,E4 0.0,E5 0.0,E6 0.0}
DECL FDAT FP12={TOOL_NO 10,BASE_NO 0,IPO_FRAME #BASE,POINT2[] " ",TQ_STATE FALSE}
DECL LDAT LCPDAT11={VEL 2.0,ACC 100.0,APO_DIST 0.0,APO_FAC 50.0,AXIS_VEL 100.0,AXIS_ACC 100.0,ORI_TYP #VAR,CIRC_TYP #BASE,JERK_FAC 50.0,GEAR_JERK 50.0,EXAX_IGN 0}
DECL E6POS XP14={X -3793.68091,Y -5863.93994,Z 1686.84204,A -114.976196,B 89.1287308,C -26.8414001,S 6,T 50,E1 -4892.8208,E2 0.0,E3 0.0,E4 0.0,E5 0.0,E6 0.0}
DECL FDAT FP14={TOOL_NO 10,BASE_NO 0,IPO_FRAME #BASE,POINT2[] " ",TQ_STATE FALSE}
DECL LDAT LCPDAT13={VEL 2.0,ACC 100.0,APO_DIST 0.0,APO_FAC 50.0,AXIS_VEL 100.0,AXIS_ACC 100.0,ORI_TYP #VAR,CIRC_TYP #BASE,JERK_FAC 50.0,GEAR_JERK 50.0,EXAX_IGN 0}
DECL GRP_TYP GGDAT3={G_APO #NO,GRP_TIME 0.200000003,CTRL #OFF,DLY 0,DST 1}
DECL GRP_TYP GGDAT4={G_APO #NO,GRP_TIME 0.200000003,CTRL #OFF,DLY 0,DST 1}
DECL GRP_TYP GGDAT5={G_APO #NO,GRP_TIME 0.200000003,CTRL #OFF,DLY 0,DST 1}
DECL GRP_TYP GGDAT28={G_APO #NO,GRP_TIME 0.200000003,CTRL #OFF,DLY 0,DST 1}
DECL GRP_TYP GGDAT29={G_APO #NO,GRP_TIME 0.200000003,CTRL #OFF,DLY 0,DST 1}
DECL GRP_TYP GGDAT26={G_APO #NO,GRP_TIME 0.200000003,CTRL #OFF,DLY 0,DST 1}
DECL GRP_TYP GGDAT27={G_APO #NO,GRP_TIME 0.200000003,CTRL #OFF,DLY 0,DST 1}
DECL GRP_TYP GGDAT30={G_APO #NO,GRP_TIME 0.200000003,CTRL #OFF,DLY 0,DST 1}
DECL GRP_TYP GGDAT6={G_APO #NO,GRP_TIME 0.200000003,CTRL #OFF,DLY 0,DST 1}
DECL GRP_TYP GCONT={G_APO #YES,GRP_TIME 0.0,CTRL #OFF,DLY 0,DST 0}
DECL E6POS XP17={X -358.77359,Y -4874.91406,Z 2799.07007,A 154.024002,B -58.8499794,C -75.7817383,S 6,T 18,E1 -3477.55103,E2 0.0,E3 0.0,E4 0.0,E5 0.0,E6 0.0}
DECL FDAT FP17={TOOL_NO 8,BASE_NO 0,IPO_FRAME #BASE,POINT2[] " ",TQ_STATE FALSE}
DECL PDAT PPDAT10={VEL 100.0,ACC 100.0,APO_DIST 10.0,APO_MODE #CDIS}
DECL PDAT PPDAT11={VEL 100.0,ACC 100.0,APO_DIST 100.0,APO_MODE #CDIS}
DECL E6POS XP18={X 10.7094097,Y -2837.7749,Z 2797.60205,A -29.1030102,B -57.9046783,C 123.9198,S 2,T 10,E1 -1390.39697,E2 0.0,E3 0.0,E4 0.0,E5 0.0,E6 0.0}
DECL FDAT FP18={TOOL_NO 8,BASE_NO 0,IPO_FRAME #BASE,POINT2[] " ",TQ_STATE FALSE}
DECL E6POS XP20={X -3804.75708,Y -5834.06201,Z 1682.58301,A -171.014099,B 89.4823608,C -83.3636093,S 6,T 50,E1 -4828.73193,E2 0.0,E3 0.0,E4 0.0,E5 0.0,E6 0.0}
DECL FDAT FP20={TOOL_NO 10,BASE_NO 0,IPO_FRAME #BASE,POINT2[] " ",TQ_STATE FALSE}
DECL PDAT PPDAT13={VEL 100.0,ACC 50.0,APO_DIST 20.0,APO_MODE #CDIS}
DECL E6POS XP21={X -3804.74292,Y -5834.10986,Z 1682.60706,A -170.702301,B 89.4826736,C -83.0520935,S 6,T 50,E1 -4828.73096,E2 0.0,E3 0.0,E4 0.0,E5 0.0,E6 0.0}
DECL FDAT FP21={TOOL_NO 10,BASE_NO 0,IPO_FRAME #BASE,POINT2[] " ",TQ_STATE FALSE}
DECL PDAT PPDAT14={VEL 100.0,ACC 50.0,APO_DIST 20.0,APO_MODE #CDIS}
DECL PDAT PP_OLP15={VEL 100.0,ACC 50.0,APO_DIST 30.0,APO_MODE #CDIS}
DECL E6POS Xl031={X -2716.59692,Y -4314.85889,Z 1766.00305,A -99.9313431,B 83.240097,C 22.9195004,S 6,T 50,E1 -3600.0,E2 0.0,E3 0.0,E4 0.0,E5 0.0,E6 0.0}
DECL FDAT Fl031={TOOL_NO 10,BASE_NO 0,IPO_FRAME #BASE,POINT2[] " "}
DECL PDAT PP_OLP16={VEL 100.0,ACC 50.0,APO_DIST 30.0,APO_MODE #CDIS}
DECL E6POS Xl036={X -3454.84399,Y -4870.63379,Z 1739.21497,A -94.3164673,B 83.0381088,C 8.50661659,S 6,T 50,E1 -4499.99902,E2 0.0,E3 0.0,E4 0.0,E5 0.0,E6 0.0}
DECL FDAT Fl036={TOOL_NO 10,BASE_NO 0,IPO_FRAME #BASE,POINT2[] " "}
ENDDAT
